{attribute 'qualified_only'}
TYPE SlaveInfoSteps :
(  
	Begin,
  FetchSlaveNames,
  End
);
END_TYPE

(* stored: Version 1.1.0.1
   DUT SlaveInfoSteps: Id {07555201-a33a-4800-9dd8-7add35bd2b97} *)
